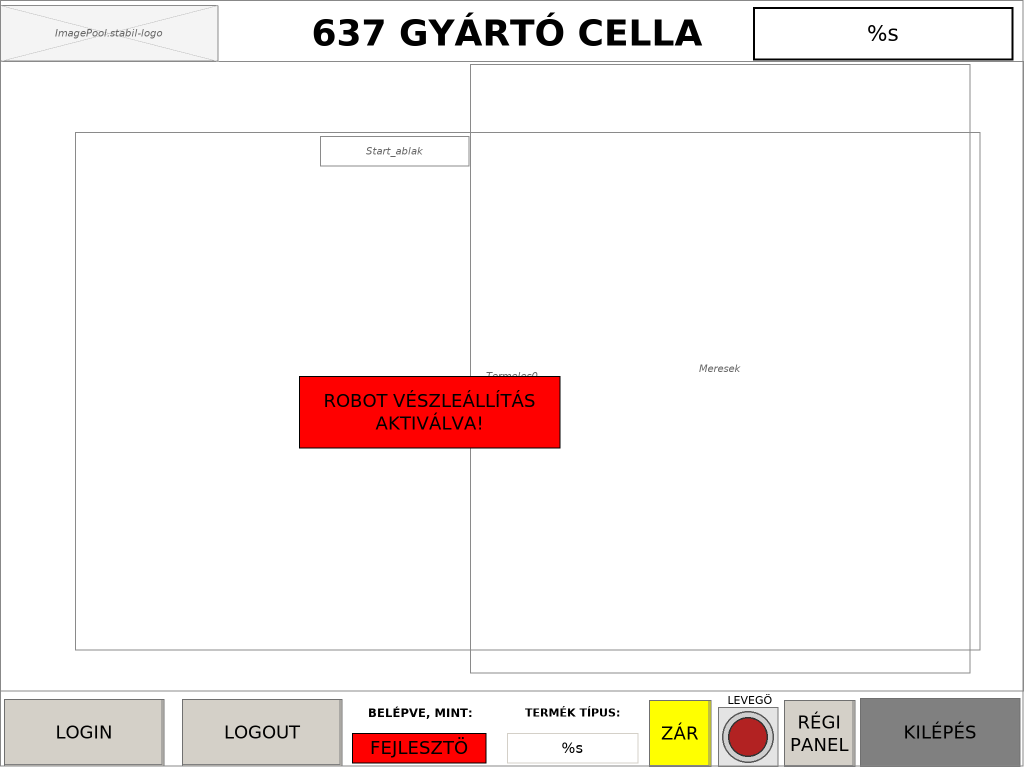
VISUALIZATION Visualization_new  // 1024x767
    TabControl (0,61 1024x630), invisible if: GVL.bSystemNotStarted, frame switch variable: GVL.iFoLapozo
        shows Termeles0()
        shows Beallitasok()
        shows Szerviz()
        shows TempJozsi()
        shows TempPisti()
        shows Laser()
        shows HegesztesGrafikon()
        [0]: TabTitle=Termelés
        [1]: TabTitle=Beállítások
        [2]: TabTitle=Szervíz
        [3]: TabTitle=Józsi
        [4]: TabTitle=Pisti
        [5]: TabTitle=Lézer
        [6]: TabTitle=Útmérés
    Image (0,5 218x56), image: ImagePool.stabil-logo
    Label (303,9 408x48), "637 GYÁRTÓ CELLA"
    RoundedRectangle (753,7 260x53), "%s", text variable: GVL.sDateTime
    Button (4,699 160x67), "LOGIN"
        OnMouseClick: VisuUserMgmt Type=Login
    Button (860,698 160x69), "KILÉPÉS"
        OnMouseClick: execute { INIT.bStartShutDown:=TRUE; }
    Button (784,700 71x67), "RÉGI PANEL", invisible if: GVL.bSystemNotStarted
        OnMouseClick: execute { GVL.bRegiFelulet:=TRUE; }
    Button (649,700 62x67), "ZÁR", colour toggle: NOT GVL.bBiztonsagiZarBe, pressed state: GVL.bBiztonsagiZarBe, invisible if: NOT INIT.bRobotKesz
        toggle GVL.bBiztonsagiZarGomb
    Label (518,698 110x30), "TERMÉK TÍPUS:"
    Textfield (507,733 131x30), "%s", text variable: GVL.sProductType, colour toggle: NOT GVL.bProductTypeOK
        OnMouseClick: write the text variable via Edit
    Group (718,691 60x76)
        Label (2,0 55x19), "LEVEGÖ"
        PushSwitch (0,16 60x60), variable: MAIN.bLevego, behaviour: TOGGLE, style: Switch-PushSwitch-Red
    Frame (470,64 500x609), invisible if: GVL.bMeresiEredmenyekRejtve
        shows Meresek()
    Frame (75,132 905x518), invisible if: GVL.bKameraEredmenyekRejtve
        shows Kamera()
    Frame (320,136 149x30), invisible if: GVL.bSystemStarted, input disabled if: GVL.bSystemStarted
        shows Start_ablak()
    Button (182,699 160x67), "LOGOUT"
        OnMouseClick: VisuUserMgmt Type=Logout
    Label (362,698 117x30), "BELÉPVE, MINT:"
    Rectangle (352,733 134x30), "SZERVÍZ"
    Rectangle (352,733 134x30), "FEJLESZTÖ"
    RoundedRectangle (299,376 261x72), "ROBOT VÉSZLEÁLLÍTÁS AKTIVÁLVA!", invisible if: NOT RobotProcess.baStatus[6]
END_VISUALIZATION

(* stored: Version 1.1.0.1, ProductVersion 3.1.4024.11
   Visu Visualization_new: Id {8700da3a-6aa4-49bb-94a7-c768f6bebfe3} *)
